// TIA Portal V20 export
DATA_BLOCK "HmiInterface"   // DB68
// stored: Access Published, MemoryReserve 100, Namespace Unit1.Em7
   VAR
      em : "LAF_typeEmInterface";
      hotPressRight : "LER_typeSequenceInterface";
      cmHotPressRightSafetyPin : "LBC_typeDigitalSignalInterface";
      cmHotPressRightJRDetect : "LBC_typeDigitalSignalInterface";
      cmHotPressRightStageLiftFrontUpDown : "LBC_typeTwoWayActuatorInterface";
      cmHotPressRightStageLiftRearUpDown : "LBC_typeTwoWayActuatorInterface";
      cmHotPressRightStageLiftAllUpDown : "LBC_typeTwoWayActuatorInterface";
      cmHotPressRightServoPress : "LER_typeServoPressInterface";
      cmHotPressRightTemperature : "LER_typeHeaterInterface";
   END_VAR
   VAR RETAIN
      cmHotPressRightHistory : "LER_typeServoPressHistory";
   END_VAR
   VAR
      intCondition : "Unit1.Em7.typeIntConditionHmiInterface";
   END_VAR
BEGIN
   cmHotPressRightTemperature.configuration.E5CC[1..5].Temp_AlarmValue1 := 1;
   cmHotPressRightTemperature.configuration.E5CC[1..5].Temp_AlarmValue1_UpperLimit := 2;
   cmHotPressRightTemperature.configuration.E5CC[1..5].Temp_AlarmValue1_LowerLimit := -2;
   cmHotPressRightTemperature.configuration.E5CC[1..5].Temp_AlarmValue2 := 3;
   cmHotPressRightTemperature.configuration.E5CC[1..5].Temp_AlarmValue2_UpperLimit := 2;
   cmHotPressRightTemperature.configuration.E5CC[1..5].Temp_AlarmValue2_LowerLimit := -2;
   cmHotPressRightTemperature.configuration.E5CC[1..5].Temp_Upper_Limit_Temp := 50;
   cmHotPressRightTemperature.configuration.E5CC[1..5].Temp_Lower_Limit_Temp := 20;
   cmHotPressRightTemperature.configuration.E5CC[1..5].Temp_MC_Off_Value := 0;
   cmHotPressRightTemperature.configuration.E5CC[1..5].Temp_Upper_Complete_Range := 1;
   cmHotPressRightTemperature.configuration.E5CC[1..5].Temp_Lower_Complete_Range := -1;
END_DATA_BLOCK
